(* IEC 61131-3 sources: Temperature-Cabinet-Control-Automation/temperature swing integration/codesys, 5 files *)

(* ---- E_TemperatureSwingState.st ---- *)
{attribute 'qualified_only'}
TYPE E_TemperatureSwingState :
(
    IDLE                := 0,
    START               := 1,
    RAMP                := 2,
    MONITOR_RATE         := 3,
    APPROACH_EXTREME     := 4,
    VERIFY_EXTREME        := 5,
    STABILISE            := 6,
    OVERSHOOT_CHECK       := 7,
    HOLD_EXTREME          := 8,
    RETURN                := 9,
    RETURN_STABILISE      := 10,
    CYCLE_COMPLETE         := 11
);
END_TYPE

(* ---- GVL_TemperatureSwing.st ---- *)
{attribute 'qualified_only'}
VAR_GLOBAL
    // ========================================================================
    // TEMPERATURE SWING TEST VARIABLES
    // See docs/GVL_TemperatureSwing_Variables.md for the field-by-field reference
    // ========================================================================

    // --- Program selection and control ---
    xProgram_TemperatureSwing          : BOOL;
    xTemperatureSwing_Start            : BOOL;
    xTemperatureSwing_Stop             : BOOL;
    xTemperatureSwing_Active           : BOOL;

    // --- Operator input (Start Dialog) ---
    rTemperatureSwing_Extreme          : REAL;
    rTemperatureSwing_PressureMode     : REAL;   // 0 / 50 / 75 / 100
    rTemperatureSwing_HoldTime         : REAL;   // minutes

    // --- State machine ---
    iTemperatureSwing_CurrentState     : INT := 0; // see E_TemperatureSwingState

    // --- Temperature monitoring ---
    rBodyTemp_Current                  : REAL;
    rBodyTemp_Previous_60s             : REAL;
    rTemperatureSwing_Rate             : REAL;
    xTemperatureSwing_RateCheckPassed  : BOOL;
    iTemperatureSwing_ConsecutivePassWindows : INT;
    xTemperatureSwing_UsingFallbackChannel   : BOOL;

    // --- Extreme / overshoot detection ---
    xTemperatureSwing_ExtremeReached   : BOOL;
    rTemperatureSwing_Overshoot        : REAL;
    rTemperatureSwing_MaxOvershoot     : REAL;
    xTemperatureSwing_OvershootExceeded : BOOL;

    // --- Pressure control ---
    rTemperatureSwing_EstablishedPressure : REAL;
    xTemperatureSwing_PressureReady    : BOOL;
    rTemperatureSwing_PressureError    : REAL;

    // --- Timers ---
    iTemperatureSwing_HoldTimer        : INT;    // seconds
    tTemperatureSwing_RampStartTime    : TIME;
    tTemperatureSwing_CycleStartTime   : TIME;

    // --- Logging ---
    sTemperatureSwing_LogFile          : STRING(255);
    xTemperatureSwing_LoggingActive    : BOOL;
    iTemperatureSwing_DataPoints       : INT;

    // --- Errors ---
    xTemperatureSwing_Error            : BOOL;
    sTemperatureSwing_ErrorMessage     : STRING(255);
    iTemperatureSwing_ErrorCode        : INT;
END_VAR

(* ---- FB_Temperature_Swing.st ---- *)
FUNCTION_BLOCK FB_Temperature_Swing
// ============================================================================
// DRAFT V2 — structure only, states not yet implemented.
// Confirmed against real project code (FB_Hold, FB_Apply_Test_Pressure,
// FB_Pressure_Release, FB_EStop, FB_CSV_Handler):
//   - Isolate convention: TRUE = closed, FALSE = open ("Normally Open").
//   - FB_Apply_Test_Pressure has no inputs, fills via doUpstream, closes once
//     at the high alarm — it never re-opens, so it cannot relieve pressure
//     that keeps rising afterwards (e.g. from heating). No existing FB does
//     that either; the vent logic below is new, built on the same bang-bang
//     convention as FB_Apply_Test_Pressure / FB_Pressure_Release.
//   - CSV recording starts/stops automatically off GVL.xStart / GVL.xSave
//     (FB_CSV_Handler.IDLE) — nothing to trigger explicitly here.
//   - Monitor channel: reuse GVL.iMainChannelIndex directly, same as FB_Hold.
//   - Hold period: INT minutes, converted with DINT_TO_TIME(*60000), same as
//     FB_Hold's iHoldPeriod — not TIME, not REAL.
// ============================================================================
VAR_INPUT
	xStart					: BOOL;
	iStep					: INT;
END_VAR
VAR_OUTPUT
	xDone					: BOOL;
END_VAR
VAR
	fbApplyPressure			: FB_Apply_Test_Pressure;   // no inputs, call every scan
	fbTarget				: FB_Temperature_Target;    // ramp direction / reached helper
	rMonitorValue			: LREAL;
	rCurrentRate			: LREAL;
	RateWindowTimer			: TON;                      // 30 s rate window
	HoldTimer				: TON;
	rRateWindowStart		: LREAL;                    // temperature at window start
	tScanCycle				: TIME := T#100MS;          // assumed scan time for rate calc
END_VAR

// ============================================================================
// CONTINUOUS — runs every scan from state 1 onward, independent of state
// ============================================================================
IF GVL.iTestPressure > 0 AND iStep >= 1 THEN
	// Fill: existing FB, closes doUpstream once at the high alarm.
	fbApplyPressure();

	// Relieve: NEW logic, not an existing FB. Same bang-bang convention —
	// open downstream while over the high alarm (thermal expansion venting),
	// close once back in band. Modelled on FB_Pressure_Release's pattern but
	// against the upper alarm instead of a low one.
	IF GVL.alrChannelReading[1] > GVL.aiAlarms[1] THEN
		GVL.doDownstream := FALSE; // open, vent excess
	ELSE
		GVL.doDownstream := TRUE;  // closed, hold
	END_IF
END_IF

// Monitor channel + rate, sampled continuously so the value is already valid
// when the stabilisation state is entered.
rMonitorValue := GVL.alrChannelReading[GVL.iMainChannelIndex];

// Rate calculation: updated every 30 s window cycle in state 6.
// Rate = (delta over 30 s) / 0.5 min = delta * 2, in °C/min.
// Window start is captured when RateWindowTimer resets; rate is calculated
// when the next window completes (checked in state 6).
IF NOT RateWindowTimer.Q THEN
	// Window in progress: rate from previous complete window remains valid
	rCurrentRate := (rMonitorValue - rRateWindowStart) * 2.0; // delta * (1 min / 0.5 min)
ELSE
	// Window just completed: capture this reading for next window's calculation
	rRateWindowStart := rMonitorValue;
END_IF

// ============================================================================
// STATE MACHINE
// ============================================================================
CASE iStep OF

	// 0: IDLE
	// Does: wait for operator Start.
	// Next: xStart -> 1.
	// Reuse: GVL.sPrompt + xStart, same as FB_Hold step 0.
	0:
		GVL.sPrompt := 'Program: Temperature Swing. Press Start to begin.';
		IF xStart THEN
			iStep := 1;
		END_IF

	// 1: STARTUP
	// Does: reset run data. If Test Pressure = 0, set the vent-safe default
	// (Upstream closed, Downstream open). CSV recording starts automatically
	// off GVL.xStart (FB_CSV_Handler) — nothing to call here.
	// Next: Test Pressure = 0 -> 3, otherwise -> 2.
	// Reuse: FB_Hold / FUN_Program_Startup pattern for isolate defaults.
	1:
		xDone := FALSE;
		IF GVL.iTestPressure = 0 THEN
			GVL.doUpstream := TRUE;    // closed
			GVL.doDownstream := FALSE; // open — nothing to build, vent path clear
			iStep := 3;
		ELSE
			iStep := 2;
		END_IF

	// 2: ESTABLISH_PRESSURE
	// Does: wait for the chamber to reach the alarm pressure before heating
	// starts. Fill/relieve logic above is already running.
	// Next: fbApplyPressure.xDone -> 3.
	// Reuse: FB_Apply_Test_Pressure.
	2:
		IF fbApplyPressure.xDone THEN
			iStep := 3;
		END_IF

	// 3: CABINET_START
	// Does: start the temperature cabinet.
	// Next: start commanded -> 4.
	// Reuse: GVL_HMI.xStartPulse relay path (EL2869 -> Omron CPM1A).
	3:
		GVL_HMI.xStartPulse := TRUE;
		iStep := 4;

	// 4: SEND_SETPOINT
	// Does: write the operator setpoint to the cabinet and arm fbTarget with
	// the ramp direction.
	// Next: write confirmed -> 5.
	// Reuse: existing Modbus TCP setpoint write/read-back path.
	4:
		fbTarget(xArm := TRUE, rSetpoint := GVL.rTemperatureSwing_Setpoint,
			rActual := rMonitorValue);
		// TODO: Modbus setpoint write to cabinet + read-back confirmation.
		// Confirm Modbus register map and implement write/read-back cycle here.
		// On confirmation, transition to state 5. On timeout/failure, route to state 9.
		iStep := 5;

	// 5: RAMP
	// Does: cabinet ramps at its own natural rate. Pressure fill/relieve runs
	// continuously above. Monitor channel shown white on the HMI.
	// Next: fbTarget.xReached -> 6.
	// Reuse: FB_Temperature_Target.
	5:
		GVL.sPrompt := 'Ramping to setpoint.';
		fbTarget(xArm := TRUE, rSetpoint := GVL.rTemperatureSwing_Setpoint,
			rActual := rMonitorValue);
		IF fbTarget.xReached THEN
			iStep := 6;
		END_IF

	// 6: STABILISE
	// Does: wait for the first 30 s window with |rate| < 0.5 degC/min.
	// Monitor channel shown orange on the HMI.
	// Next: first passing window -> 7.
	// Reuse: rate already calculated continuously above.
	6:
		GVL.sPrompt := 'Stabilising: waiting for rate below 0.5 degC/min.';
		// On first entry to this state, capture the starting temperature for rate window
		IF RateWindowTimer.IN = FALSE THEN
			rRateWindowStart := rMonitorValue;
		END_IF;
		RateWindowTimer(IN := TRUE, PT := T#30S);
		IF RateWindowTimer.Q THEN
			RateWindowTimer(IN := FALSE);
			IF ABS(rCurrentRate) < 0.5 THEN
				iStep := 7;
			END_IF
		END_IF

	// 7: HOLD
	// Does: hold at setpoint for the operator-configured hold period.
	// Next: hold elapsed -> 8.
	// Reuse: FB_Hold timer pattern — INT minutes via DINT_TO_TIME(*60000).
	7:
		GVL.sPrompt := 'Holding at setpoint.';
		HoldTimer(IN := TRUE, PT := DINT_TO_TIME(GVL.iTemperatureSwing_HoldPeriod * 60000));
		IF HoldTimer.Q THEN
			HoldTimer(IN := FALSE);
			iStep := 8;
		END_IF

	// 8: COMPLETE
	// Does: leave the cabinet running at setpoint, wait for save. CSV closes
	// automatically off GVL.xSave (FB_CSV_Handler).
	// Next: GVL.xSave -> xDone, iStep := 0.
	// Reuse: FB_Hold save-then-stop pattern.
	8:
		GVL.sPrompt := 'Test complete — press End to finish.';
		IF GVL.xSave THEN
			xDone := TRUE;
			iStep := 0;
		END_IF

	// 9: ERROR
	// Does: hold the rig and wait for operator acknowledgement.
	// Next: acknowledged -> xDone, iStep := 0.
	// Reuse: FB_Hold overpressure-handling pattern. E-stop is already handled
	// centrally by ProgramSelecter / FB_EStop.
	9:
		GVL.sPrompt := 'Temperature Swing error — press Stop.';
		IF NOT xStart THEN
			xDone := TRUE;
			iStep := 0;
		END_IF

END_CASE

(* ---- FB_Temperature_Target.st ---- *)
FUNCTION_BLOCK FB_Temperature_Target
// ============================================================================
// DRAFT V2 — small reusable helper.
// Latches the ramp direction on arming, then reports when the temperature has
// reached or passed the setpoint in that direction. Keeps the heating/cooling
// comparison out of the main Temperature Swing state machine, and is reusable
// by any future program that ramps to a temperature.
// ============================================================================
VAR_INPUT
	xArm					: BOOL;     // TRUE from the setpoint write onwards
	rSetpoint				: LREAL;
	rActual					: LREAL;
END_VAR
VAR_OUTPUT
	xReached				: BOOL;
	xHeating				: BOOL;     // latched direction, for HMI/logging
END_VAR
VAR
	xArmed					: BOOL;
END_VAR

IF NOT xArm THEN
	xArmed   := FALSE;
	xReached := FALSE;
ELSE
	// Latch direction once, on the first scan after arming.
	IF NOT xArmed THEN
		xHeating := (rSetpoint > rActual);
		xArmed   := TRUE;
	END_IF

	IF xHeating THEN
		xReached := (rActual >= rSetpoint);
	ELSE
		xReached := (rActual <= rSetpoint);
	END_IF
END_IF

(* ---- FB_TemperatureSwing.st ---- *)
{attribute 'qualified_only'}
FUNCTION_BLOCK FB_TemperatureSwing
(*
    Temperature Swing test state machine — API 6A F.1.9 / F.1.10 / F.1.11.

    Reuses FB_Apply_Test_Pressure for pressure establishment and the existing
    upstream/downstream solenoid pattern for pressure maintenance during the
    ramp/hold/return. See docs/Stage2_Design_Document.md for the full design
    and state diagram.
*)
VAR_INPUT
    xEnable             : BOOL;    // TRUE while xProgram_TemperatureSwing selected
END_VAR

VAR_OUTPUT
    xSolenoid_Upstream   : BOOL;
    xSolenoid_Downstream : BOOL;
END_VAR

VAR
    fbApplyPressure      : FB_Apply_Test_Pressure;
    fbStabilisationCheck : FB_Stabilisation_Check;
    tonRateWindow        : TON;    // 60 s rate-of-change window
    tonPressureTimeout   : TON;    // 300 s pressure establishment timeout
    tonHoldTimer         : TON;
    iRateSampleIndex     : INT;
    rRateBuffer          : ARRAY[0..59] OF REAL; // 1 Hz ring buffer, 60 s deep
END_VAR

// ============================================================================
// Safety exit — valid from any state
// ============================================================================
IF xTemperatureSwing_Stop OR GVL.xAlarm_Active THEN
    iTemperatureSwing_CurrentState := E_TemperatureSwingState.IDLE;
    xTemperatureSwing_Active := FALSE;
    xSolenoid_Upstream := FALSE;
    xSolenoid_Downstream := FALSE;
    tonHoldTimer(IN := FALSE);
    IF xTemperatureSwing_LoggingActive THEN
        sTemperatureSwing_ErrorMessage := 'Aborted by operator or alarm';
        F_LogTemperatureSwingRow(sTemperatureSwing_LogFile, 'ABORTED');
        xTemperatureSwing_LoggingActive := FALSE;
    END_IF;
    RETURN;
END_IF;

// ============================================================================
// Rate-of-change sampling (1 Hz), independent of state so it is always fresh
// ============================================================================
rRateBuffer[iRateSampleIndex] := rBodyTemp_Current;
iRateSampleIndex := (iRateSampleIndex + 1) MOD 60;
rBodyTemp_Previous_60s := rRateBuffer[iRateSampleIndex]; // oldest sample = 60 s ago

tonRateWindow(IN := xTemperatureSwing_Active, PT := T#60S);
IF tonRateWindow.Q THEN
    tonRateWindow(IN := FALSE);
    rTemperatureSwing_Rate := (rBodyTemp_Current - rBodyTemp_Previous_60s); // degC/min, window = 1 min
    IF ABS(rTemperatureSwing_Rate) < 0.5 THEN
        xTemperatureSwing_RateCheckPassed := TRUE;
        iTemperatureSwing_ConsecutivePassWindows := iTemperatureSwing_ConsecutivePassWindows + 1;
    ELSE
        xTemperatureSwing_RateCheckPassed := FALSE;
        iTemperatureSwing_ConsecutivePassWindows := 0;
    END_IF;
    F_LogTemperatureSwingRow(sTemperatureSwing_LogFile, 'RATE_SAMPLE');
END_IF;

// ============================================================================
// Pressure maintenance — active in RAMP..HOLD_EXTREME, closed-loop bang-bang
// ============================================================================
IF xTemperatureSwing_PressureReady AND xTemperatureSwing_Active THEN
    rTemperatureSwing_PressureError := rTemperatureSwing_EstablishedPressure - GVL.rChamberPressure_Current;
    IF rTemperatureSwing_PressureError > 0.5 THEN
        xSolenoid_Upstream := TRUE;
        xSolenoid_Downstream := FALSE;
    ELSIF rTemperatureSwing_PressureError < -0.5 THEN
        xSolenoid_Upstream := FALSE;
        xSolenoid_Downstream := TRUE;
    ELSE
        xSolenoid_Upstream := FALSE;
        xSolenoid_Downstream := FALSE;
    END_IF;
ELSE
    xSolenoid_Upstream := FALSE;
    xSolenoid_Downstream := FALSE;
END_IF;

// ============================================================================
// State machine
// ============================================================================
CASE iTemperatureSwing_CurrentState OF

    E_TemperatureSwingState.IDLE:
        xTemperatureSwing_Active := FALSE;
        IF xEnable AND xTemperatureSwing_Start THEN
            tTemperatureSwing_CycleStartTime := GVL.tSystemTime;
            sTemperatureSwing_LogFile := F_BuildTemperatureSwingLogPath(rTemperatureSwing_Extreme);
            xTemperatureSwing_LoggingActive := TRUE;
            iTemperatureSwing_DataPoints := 0;
            rTemperatureSwing_MaxOvershoot := 0.0;
            xTemperatureSwing_OvershootExceeded := FALSE;
            iTemperatureSwing_CurrentState := E_TemperatureSwingState.START;
        END_IF;

    E_TemperatureSwingState.START:
        xTemperatureSwing_Active := TRUE;
        // Establish pressure before any ramp begins
        fbApplyPressure(
            rTargetPressure := (rTemperatureSwing_PressureMode / 100.0) * GVL.rTestProfile_Pressure,
            xStart          := TRUE);
        tonPressureTimeout(IN := TRUE, PT := T#300S);

        IF fbApplyPressure.xDone THEN
            fbApplyPressure(xStart := FALSE);
            tonPressureTimeout(IN := FALSE);
            rTemperatureSwing_EstablishedPressure := (rTemperatureSwing_PressureMode / 100.0) * GVL.rTestProfile_Pressure;
            xTemperatureSwing_PressureReady := TRUE;
            tTemperatureSwing_RampStartTime := GVL.tSystemTime;
            iTemperatureSwing_CurrentState := E_TemperatureSwingState.RAMP;
        ELSIF fbApplyPressure.xError OR tonPressureTimeout.Q THEN
            xTemperatureSwing_Error := TRUE;
            sTemperatureSwing_ErrorMessage := 'Pressure establishment failed or timed out';
            iTemperatureSwing_ErrorCode := 1001;
            F_LogTemperatureSwingRow(sTemperatureSwing_LogFile, 'ERROR_PRESSURE');
            iTemperatureSwing_CurrentState := E_TemperatureSwingState.IDLE;
        END_IF;

    E_TemperatureSwingState.RAMP:
        GVL.rCabinetSetpoint_Command := rTemperatureSwing_Extreme; // drives cabinet via existing setpoint-write path
        iTemperatureSwing_CurrentState := E_TemperatureSwingState.MONITOR_RATE;

    E_TemperatureSwingState.MONITOR_RATE:
        IF iTemperatureSwing_ConsecutivePassWindows >= 2 THEN
            iTemperatureSwing_CurrentState := E_TemperatureSwingState.APPROACH_EXTREME;
        END_IF;

    E_TemperatureSwingState.APPROACH_EXTREME:
        IF ABS(rBodyTemp_Current - rTemperatureSwing_Extreme) <= 2.0 THEN
            iTemperatureSwing_CurrentState := E_TemperatureSwingState.VERIFY_EXTREME;
        END_IF;

    E_TemperatureSwingState.VERIFY_EXTREME:
        IF (rTemperatureSwing_Extreme >= 0.0 AND rBodyTemp_Current >= rTemperatureSwing_Extreme) OR
           (rTemperatureSwing_Extreme <  0.0 AND rBodyTemp_Current <= rTemperatureSwing_Extreme) THEN
            xTemperatureSwing_ExtremeReached := TRUE;
            iTemperatureSwing_CurrentState := E_TemperatureSwingState.STABILISE;
        END_IF;

    E_TemperatureSwingState.STABILISE:
        rTemperatureSwing_Overshoot := ABS(rBodyTemp_Current - rTemperatureSwing_Extreme);
        rTemperatureSwing_MaxOvershoot := MAX(rTemperatureSwing_MaxOvershoot, rTemperatureSwing_Overshoot);
        IF xTemperatureSwing_RateCheckPassed THEN
            iTemperatureSwing_CurrentState := E_TemperatureSwingState.OVERSHOOT_CHECK;
        END_IF;

    E_TemperatureSwingState.OVERSHOOT_CHECK:
        IF rTemperatureSwing_MaxOvershoot > 11.0 THEN
            xTemperatureSwing_OvershootExceeded := TRUE; // logged, non-aborting per design
            F_LogTemperatureSwingRow(sTemperatureSwing_LogFile, 'OVERSHOOT_EXCEEDED');
        END_IF;
        iTemperatureSwing_HoldTimer := TO_INT(rTemperatureSwing_HoldTime * 60.0);
        tonHoldTimer(IN := TRUE, PT := TIME_OF_DAY_TO_TIME(T#0S) + TO_TIME(iTemperatureSwing_HoldTimer * 1000));
        iTemperatureSwing_CurrentState := E_TemperatureSwingState.HOLD_EXTREME;

    E_TemperatureSwingState.HOLD_EXTREME:
        IF iTemperatureSwing_HoldTimer > 0 THEN
            iTemperatureSwing_HoldTimer := iTemperatureSwing_HoldTimer - 1; // decremented on 1 s task cycle
        ELSE
            tonHoldTimer(IN := FALSE);
            iTemperatureSwing_ConsecutivePassWindows := 0; // require fresh confirmation on the return leg
            iTemperatureSwing_CurrentState := E_TemperatureSwingState.RETURN;
        END_IF;

    E_TemperatureSwingState.RETURN:
        GVL.rCabinetSetpoint_Command := GVL.rAmbientTemperature_Reference;
        iTemperatureSwing_CurrentState := E_TemperatureSwingState.RETURN_STABILISE;

    E_TemperatureSwingState.RETURN_STABILISE:
        IF iTemperatureSwing_ConsecutivePassWindows >= 2 THEN
            iTemperatureSwing_CurrentState := E_TemperatureSwingState.CYCLE_COMPLETE;
        END_IF;

    E_TemperatureSwingState.CYCLE_COMPLETE:
        F_LogTemperatureSwingRow(sTemperatureSwing_LogFile, 'CYCLE_COMPLETE');
        xTemperatureSwing_LoggingActive := FALSE;
        xTemperatureSwing_PressureReady := FALSE;
        iTemperatureSwing_CurrentState := E_TemperatureSwingState.IDLE;

END_CASE
